FUNCTION_BLOCK FB_GCC_Test EXTENDS TcUnit.FB_TestSuite
VAR_INPUT
END_VAR
VAR_OUTPUT
END_VAR
VAR
    PG : ST_VG;
    fb_MKS355: FB_MKS355;
    //fb_MKS500: FB_MKS500;
    i_iPRESS_R AT %Q* :INT;
    cycle:INT :=0;
END_VAR

M_INIT();
M_Interlock();
//M_CheckRange();
//M_SelfProtection();
cycle:=cycle+1;

METHOD M_CheckRange
VAR
    Expected:REAL;
    Actual:REAL;
    eStateExpected: E_PressureState;
    eStateActual: E_PressureState;
END_VAR
TEST('Check_Range');
Case This^.cycle of
    12:
    THIS^.fb_MKS355.i_iPRESS_R :=  V_TO_INT(1);
    THIS^.fb_MKS355.PG.rPRESS := 1E-4;
    THIS^.fb_MKS355.PG.xPRESS_OK := TRUE;
    THIS^.fb_MKS355.M_HVE(TRUE);

    15:
    TEST('MKS355 Range Valid');
    Expected :=1E-9 ;
    eStateExpected := Valid;
    Actual := THIS^.fb_MKS355.IG.rPRESS;
    eStateActual := THIS^.fb_MKS355.IG.eState;
    AssertTrue(THIS^.fb_MKS355.IG.xPRESS_OK, 'MKS355 xPRESS_OK is set to False');
    AssertEquals(eStateExpected,eStateActual,'MKS355 eState Fail');
    AssertEquals_REAL(Expected, Actual,1E-10, 'MKS355 rPress Fail');
    TEST_FINISHED_NAMED('MKS355_Range_Valid');

    20:
	THIS^.fb_MKS355.i_iPRESS_R :=  V_TO_INT(0.001);
    TEST('MKS355 Range ValidLo');
    Expected :=1E-10;
    Actual := THIS^.fb_MKS355.IG.rPRESS;
    eStateExpected := ValidLo;
    eStateActual := THIS^.fb_MKS355.IG.eState;
    AssertTrue(THIS^.fb_MKS355.IG.xPRESS_OK, 'MKS355 xPRESS_OK is set to False');
    AssertEquals(eStateExpected,eStateActual,'MKS355 eState Fail');
    AssertEquals_REAL(Expected, Actual,1E-10, 'MKS355 rPress Fail');
    TEST_FINISHED_NAMED('MKS355_Range_ValidLo');


    24:
	THIS^.fb_MKS355.i_iPRESS_R :=  V_TO_INT(10);
    TEST('MKS355 Range Off');
    Expected :=0 ;
    eStateExpected := Off;
    Actual := THIS^.fb_MKS355.IG.rPRESS;
    eStateActual := THIS^.fb_MKS355.IG.eState;
    AssertFalse(THIS^.fb_MKS355.IG.xPRESS_OK, 'MKS355 xPRESS_OK is set to True');
    AssertEquals(eStateExpected,eStateActual,'MKS355 eState Fail');
    AssertEquals_REAL(Expected, Actual,1, 'MKS355 rPress Fail');
    TEST_FINISHED_NAMED('MKS355_Range_Off');


    25:
    This^.i_iPRESS_R :=  V_TO_INT(10);


    29:
    TEST('MKS355 Range Invalid');
    Expected :=0 ;
    eStateExpected := PressInvalid;
    Actual := This^.fb_MKS422.IG.rPRESS;
    eStateActual := This^.fb_MKS422.IG.eState;
    AssertFalse(This^.fb_MKS422.IG.xPRESS_OK, 'MKS422A xPRESS_OK is set to True');
    AssertEquals(eStateExpected,eStateActual,'MKS422A eState Fail');
    AssertEquals_REAL(Expected, Actual,1, 'MKS422A rPress Fail');
    TEST_FINISHED_NAMED('MKS422_Range_Invalid');
    TEST_FINISHED_NAMED('Check_Range');

END_CASE

THIS^.fb_MKS355(PG:=THIS^.PG, IG=>);
END_METHOD

METHOD M_INIT
VAR
END_VAR
TEST('MKS355_Startup');
THIS^.PG.rPRESS := 1E-4;
THIS^.PG.xPRESS_OK := TRUE;
THIS^.fb_MKS355(PG:=THIS^.PG, IG=>);
THIS^.fb_MKS355.M_HVE(TRUE);
IF( cycle = 1) THEN
    AssertTrue(THIS^.fb_MKS355.IG.xHV_SW, 'MKS355 xHV_SW set to False');
    AssertTrue(THIS^.fb_MKS355.IG.q_xHV_DIS, 'MKS355 q_xHV_DIS set to False');
    TEST_FINISHED_NAMED('MKS355_Startup');
End_IF;
END_METHOD

METHOD M_Interlock
VAR_INPUT
END_VAR
TEST('MKS355_Interlock_Active');
TEST('MKS355_Interlock_OK');
TEST('MKS355_Interlock_Lost');

CASE cycle OF
	
    3:
	THIS^.PG.rPRESS := 1E-1;
    THIS^.PG.xPRESS_OK := TRUE;
    AssertFalse(THIS^.fb_MKS355.IG.xHV_SW, 'MKS355 xHV_SW set to True');
    AssertFalse(THIS^.fb_MKS355.IG.q_xHV_DIS, 'MKS355 q_xHV_DIS set to True');
    TEST_FINISHED_NAMED('MKS355_Interlock_Active');

    4:
    This^.PG.rPRESS := 1E-4;
    This^.PG.xPRESS_OK := True;
    fb_MKS355.M_HVE(TRUE);

    7:
    AssertTrue(THIS^.fb_MKS355.IG.xHV_SW, 'MKS355 xHV_SW set to False');
    AssertTrue(THIS^.fb_MKS355.IG.q_xHV_DIS, 'MKS355 q_xHV_DIS set to False');
    TEST_FINISHED_NAMED('MKS355_Interlock_OK');

    8:
    This^.PG.rPRESS := 1E-1;
    This^.PG.xPRESS_OK := False;
    THIS^.fb_MKS355(PG:=THIS^.PG, IG=>);

    11:
    AssertFalse(THIS^.fb_MKS355.IG.xHV_SW, 'MKS422 xHV_SW set to True');
    AssertFalse(THIS^.fb_MKS355.IG.q_xHV_DIS, 'MKS422 q_xHV_DIS set to True');
    TEST_FINISHED_NAMED('MKS422_Interlock_Lost');
END_CASE

THIS^.fb_MKS355(PG:=THIS^.PG, IG=>);
END_METHOD

METHOD M_SelfProtection
VAR_INPUT
END_VAR
// Switching the Cold cathode backon
TEST('MKS355_Interlock_OK_1');
This^.PG.rPRESS := 1E-4;
This^.PG.xPRESS_OK := True;
fb_MKS355.M_HVE(TRUE);
THIS^.fb_MKS355(PG:=THIS^.PG, IG=>);
AssertTrue(THIS^.fb_MKS355.IG.xHV_SW, 'MKS355 xHV_SW set to False');
AssertFalse(THIS^.fb_MKS355.IG.q_xHV_DIS, 'MKS355 q_xHV_DIS set to True');
TEST_FINISHED_NAMED('MKS355_Interlock_OK_1');

TEST('MKS355_Self_Protection');
This^.PG.rPRESS := 1E-3;
This^.PG.xPRESS_OK := TRUE;
THIS^.fb_MKS355(PG:=THIS^.PG, IG=>);
AssertFalse(THIS^.fb_MKS355.IG.xHV_SW, 'MKS355 xHV_SW set to True');
AssertTrue(THIS^.fb_MKS355.IG.q_xHV_DIS, 'MKS355 q_xHV_DIS set to False');
TEST_FINISHED_NAMED('MKS355_Self_Protection');
END_METHOD

END_FUNCTION_BLOCK

(* stored: Version 1.1.0.1
   POU FB_GCC_Test: Id {abe007c5-97e2-4f83-88a7-7230dad873a3}, SpecialFunc None
   Method M_CheckRange: Id {1ce3796c-9d57-423a-81de-918c6cc47319}
   Method M_INIT: Id {6a239255-8bd8-42eb-b1a0-2dca15c1db92}
   Method M_Interlock: Id {376a3c27-9e60-4e4c-aaa9-e38bd67d3a7b}
   Method M_SelfProtection: Id {ee508d43-9bf6-4fa4-a8d8-d9a6f8404bfe} *)
